// TIA Portal V19 export
TYPE "TrkMng_Move"
// stored: Access Published
   STRUCT
      SelButton : Bool;
      PasteButton : Bool;
      DeleteButton : Bool;
      InfoButton : Bool;
      PasteButton_Visibile : Bool;
      DeleteButton_Visibile : Bool;
      SelectButton_Visibile : Bool;
      SelectButton_Selected : Bool;
   END_STRUCT;
END_TYPE
